PROGRAM testProg
VAR
    myFirstSlits : FB_SlitPair;

END_VAR

GVL.astAxes[1].stConfig.eHomeSeq:=E_HomingRoutines.eHomeToRef_Bwd;
GVL.astAxes[1].stConfig.fHomePosition:=-30;
GVL.astAxes[2].stConfig.eHomeSeq:=E_HomingRoutines.eHomeToRef_Fwd;
GVL.astAxes[2].stConfig.fHomePosition:=30;

myFirstSlits(iBladeNegative:=1,iBladePositive:=2, iGapSize:=3, iGapCentre:=4);

END_PROGRAM

(* stored: Version 1.1.0.1, ProductVersion 3.1.4024.5
   POU testProg: Id {6b742e2c-3720-4a26-aa80-15486c69d838}, SpecialFunc None *)
